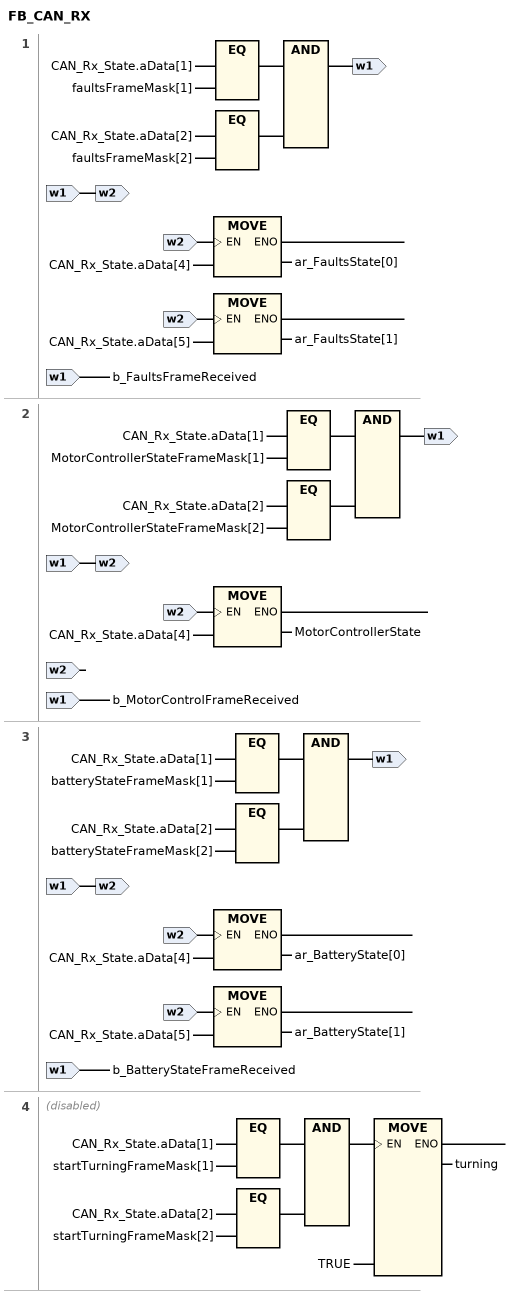
// NETWORK 1
_w1 := CAN_Rx_State.aData[1] = faultsFrameMask[1] AND CAN_Rx_State.aData[2] = faultsFrameMask[2];
_rt1(CLK := _w1);
IF _rt1.Q THEN ar_FaultsState[0] := CAN_Rx_State.aData[4]; END_IF
_rt2(CLK := _w1);
IF _rt2.Q THEN ar_FaultsState[1] := CAN_Rx_State.aData[5]; END_IF
b_FaultsFrameReceived := _w1;

// NETWORK 2
_w2 := CAN_Rx_State.aData[1] = MotorControllerStateFrameMask[1] AND CAN_Rx_State.aData[2] = MotorControllerStateFrameMask[2];
_rt3(CLK := _w2);
IF _rt3.Q THEN MotorControllerState := CAN_Rx_State.aData[4]; END_IF
b_MotorControlFrameReceived := _w2;

// NETWORK 3
_w3 := CAN_Rx_State.aData[1] = batteryStateFrameMask[1] AND CAN_Rx_State.aData[2] = batteryStateFrameMask[2];
_rt4(CLK := _w3);
IF _rt4.Q THEN ar_BatteryState[0] := CAN_Rx_State.aData[4]; END_IF
_rt5(CLK := _w3);
IF _rt5.Q THEN ar_BatteryState[1] := CAN_Rx_State.aData[5]; END_IF
b_BatteryStateFrameReceived := _w3;

// NETWORK 4 (disabled)
// _rt6(CLK := CAN_Rx_State.aData[1] = startTurningFrameMask[1] AND CAN_Rx_State.aData[2] = startTurningFrameMask[2]);
// IF _rt6.Q THEN turning := TRUE; END_IF

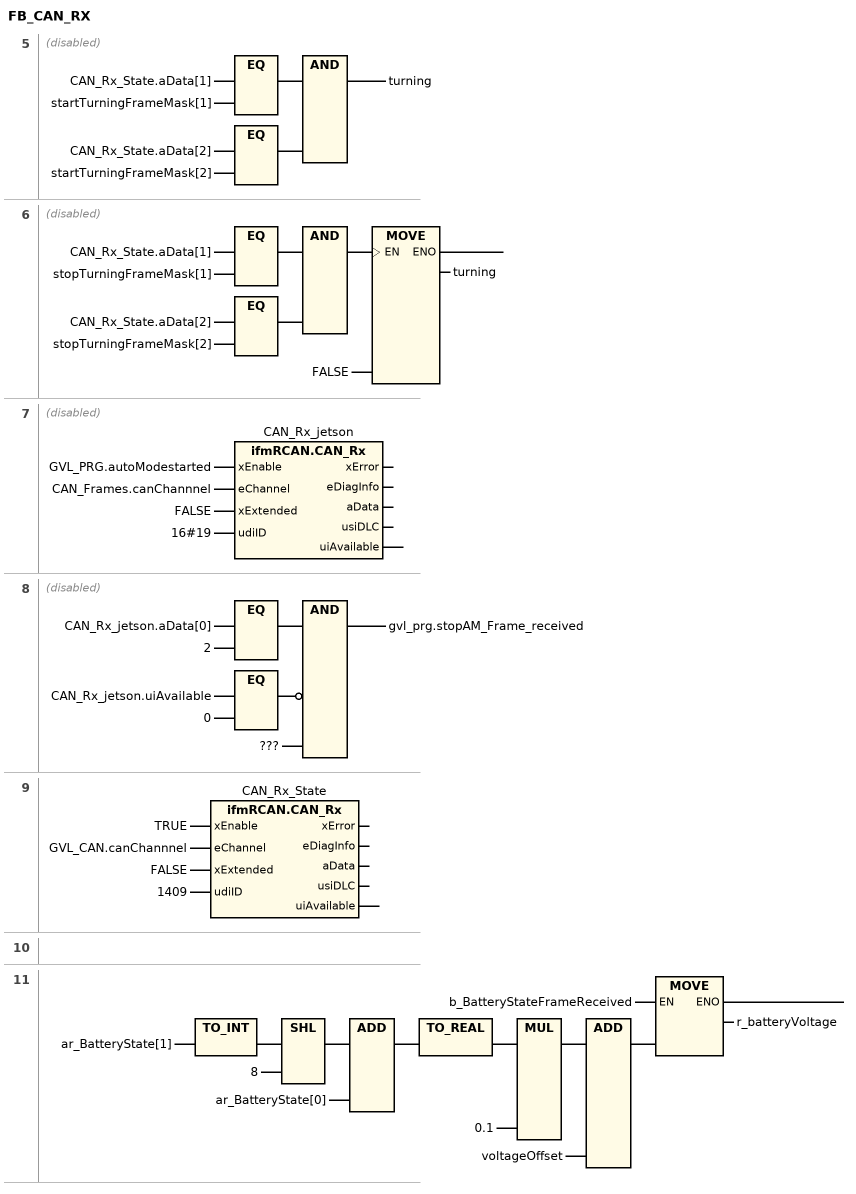
// NETWORK 5 (disabled)
// turning := CAN_Rx_State.aData[1] = startTurningFrameMask[1] AND CAN_Rx_State.aData[2] = startTurningFrameMask[2];

// NETWORK 6 (disabled)
// _rt7(CLK := CAN_Rx_State.aData[1] = stopTurningFrameMask[1] AND CAN_Rx_State.aData[2] = stopTurningFrameMask[2]);
// IF _rt7.Q THEN turning := FALSE; END_IF

// NETWORK 7 (disabled)
// CAN_Rx_jetson(
//     xEnable := GVL_PRG.autoModestarted,
//     eChannel := CAN_Frames.canChannnel,
//     xExtended := FALSE,
//     udiID := 16#19); // ifmRCAN.CAN_Rx

// NETWORK 8 (disabled)
// gvl_prg.stopAM_Frame_received := CAN_Rx_jetson.aData[0] = 2 AND NOT (CAN_Rx_jetson.uiAvailable = 0) AND ???;

// NETWORK 9
CAN_Rx_State(xEnable := TRUE, eChannel := GVL_CAN.canChannnel, xExtended := FALSE, udiID := 1409); // ifmRCAN.CAN_Rx

// NETWORK 10

// NETWORK 11
IF b_BatteryStateFrameReceived THEN
    r_batteryVoltage := TO_REAL(SHL(TO_INT(ar_BatteryState[1]), 8) + ar_BatteryState[0]) * 0.1 + voltageOffset;
END_IF

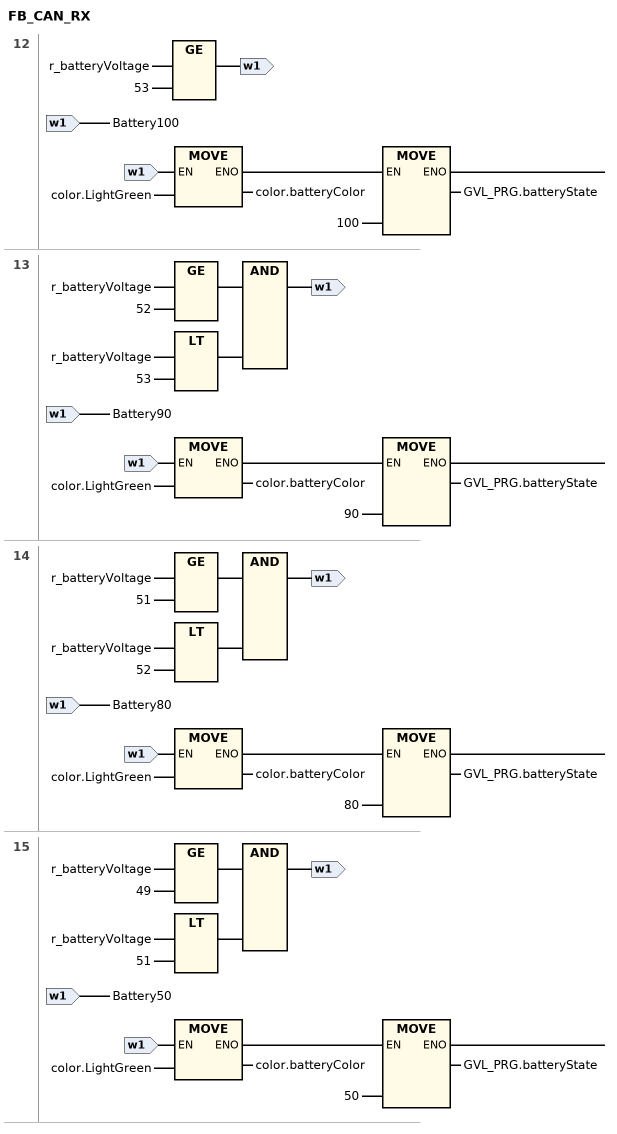
// NETWORK 12
_w4 := r_batteryVoltage >= 53;
Battery100 := _w4;
IF _w4 THEN color.batteryColor := color.LightGreen; END_IF
IF _w4 THEN GVL_PRG.batteryState := 100; END_IF

// NETWORK 13
_w5 := r_batteryVoltage >= 52 AND r_batteryVoltage < 53;
Battery90 := _w5;
IF _w5 THEN color.batteryColor := color.LightGreen; END_IF
IF _w5 THEN GVL_PRG.batteryState := 90; END_IF

// NETWORK 14
_w6 := r_batteryVoltage >= 51 AND r_batteryVoltage < 52;
Battery80 := _w6;
IF _w6 THEN color.batteryColor := color.LightGreen; END_IF
IF _w6 THEN GVL_PRG.batteryState := 80; END_IF

// NETWORK 15
_w7 := r_batteryVoltage >= 49 AND r_batteryVoltage < 51;
Battery50 := _w7;
IF _w7 THEN color.batteryColor := color.LightGreen; END_IF
IF _w7 THEN GVL_PRG.batteryState := 50; END_IF

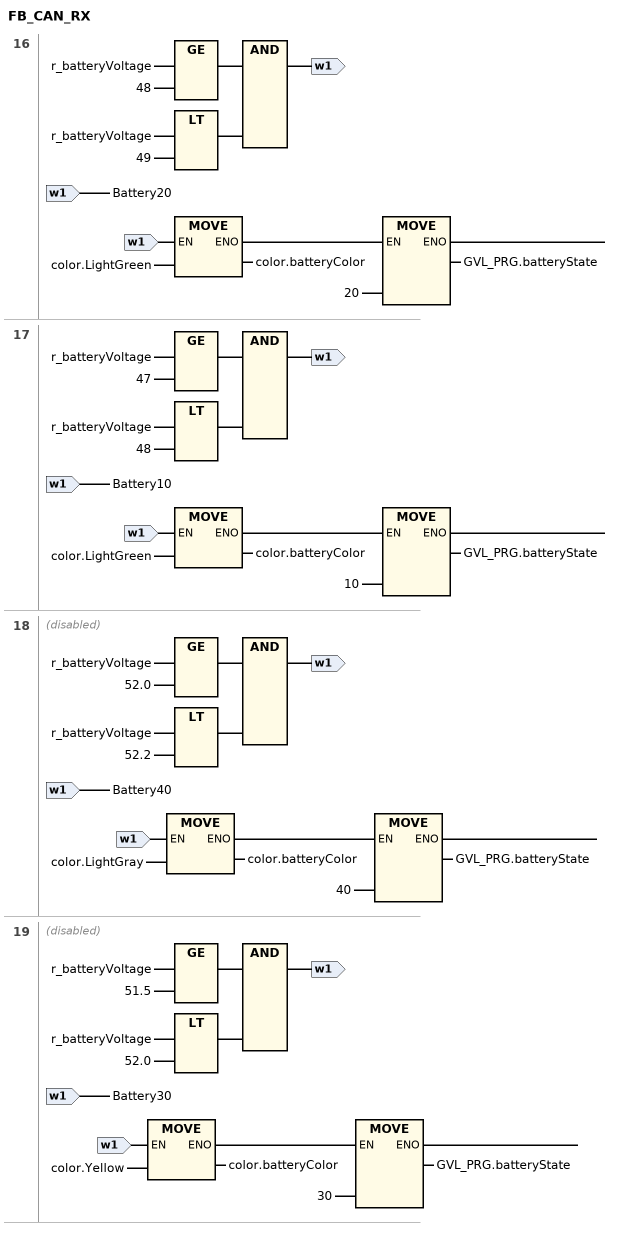
// NETWORK 16
_w8 := r_batteryVoltage >= 48 AND r_batteryVoltage < 49;
Battery20 := _w8;
IF _w8 THEN color.batteryColor := color.LightGreen; END_IF
IF _w8 THEN GVL_PRG.batteryState := 20; END_IF

// NETWORK 17
_w9 := r_batteryVoltage >= 47 AND r_batteryVoltage < 48;
Battery10 := _w9;
IF _w9 THEN color.batteryColor := color.LightGreen; END_IF
IF _w9 THEN GVL_PRG.batteryState := 10; END_IF

// NETWORK 18 (disabled)
// _w10 := r_batteryVoltage >= 52.0 AND r_batteryVoltage < 52.2;
// Battery40 := _w10;
// IF _w10 THEN color.batteryColor := color.LightGray; END_IF
// IF _w10 THEN GVL_PRG.batteryState := 40; END_IF

// NETWORK 19 (disabled)
// _w11 := r_batteryVoltage >= 51.5 AND r_batteryVoltage < 52.0;
// Battery30 := _w11;
// IF _w11 THEN color.batteryColor := color.Yellow; END_IF
// IF _w11 THEN GVL_PRG.batteryState := 30; END_IF

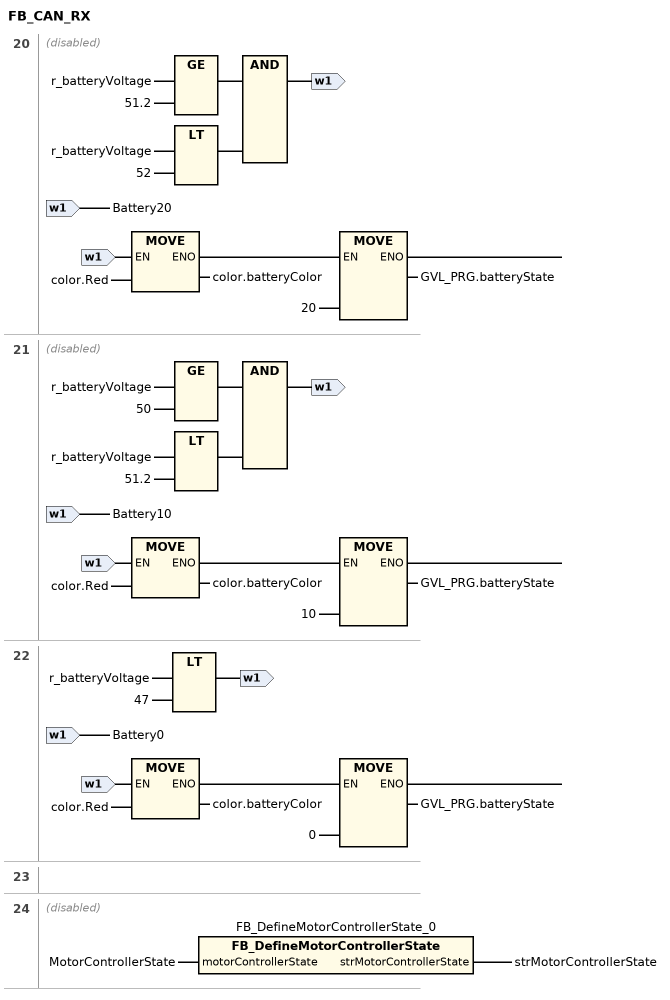
// NETWORK 20 (disabled)
// _w12 := r_batteryVoltage >= 51.2 AND r_batteryVoltage < 52;
// Battery20 := _w12;
// IF _w12 THEN color.batteryColor := color.Red; END_IF
// IF _w12 THEN GVL_PRG.batteryState := 20; END_IF

// NETWORK 21 (disabled)
// _w13 := r_batteryVoltage >= 50 AND r_batteryVoltage < 51.2;
// Battery10 := _w13;
// IF _w13 THEN color.batteryColor := color.Red; END_IF
// IF _w13 THEN GVL_PRG.batteryState := 10; END_IF

// NETWORK 22
_w14 := r_batteryVoltage < 47;
Battery0 := _w14;
IF _w14 THEN color.batteryColor := color.Red; END_IF
IF _w14 THEN GVL_PRG.batteryState := 0; END_IF

// NETWORK 23

// NETWORK 24 (disabled)
// FB_DefineMotorControllerState_0(motorControllerState := MotorControllerState); // FB_DefineMotorControllerState
// strMotorControllerState := FB_DefineMotorControllerState_0.strMotorControllerState;

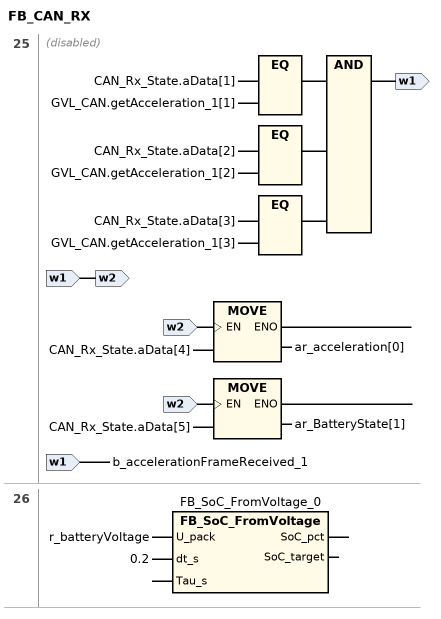
// NETWORK 25 (disabled)
// _w15 := CAN_Rx_State.aData[1] = GVL_CAN.getAcceleration_1[1] AND CAN_Rx_State.aData[2] = GVL_CAN.getAcceleration_1[2] AND CAN_Rx_State.aData[3] = GVL_CAN.getAcceleration_1[3];
// _rt8(CLK := _w15);
// IF _rt8.Q THEN ar_acceleration[0] := CAN_Rx_State.aData[4]; END_IF
// _rt9(CLK := _w15);
// IF _rt9.Q THEN ar_BatteryState[1] := CAN_Rx_State.aData[5]; END_IF
// b_accelerationFrameReceived_1 := _w15;

// NETWORK 26
FB_SoC_FromVoltage_0(U_pack := r_batteryVoltage, dt_s := 0.2); // FB_SoC_FromVoltage

END_FUNCTION_BLOCK

// Device/Application/FBs/FB_DefineMotorControllerState
FUNCTION_BLOCK FB_DefineMotorControllerState
VAR_INPUT
	motorControllerState: BYTE;
END_VAR
VAR_OUTPUT
	strMotorControllerState: STRING(100);
END_VAR
VAR
	FB_ByteToBoolArray_MotorControl: FB_ByteToBoolArray;
END_VAR

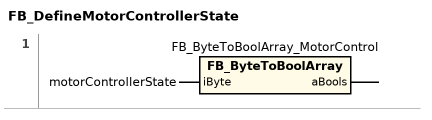
// NETWORK 1
FB_ByteToBoolArray_MotorControl(iByte := motorControllerState); // FB_ByteToBoolArray

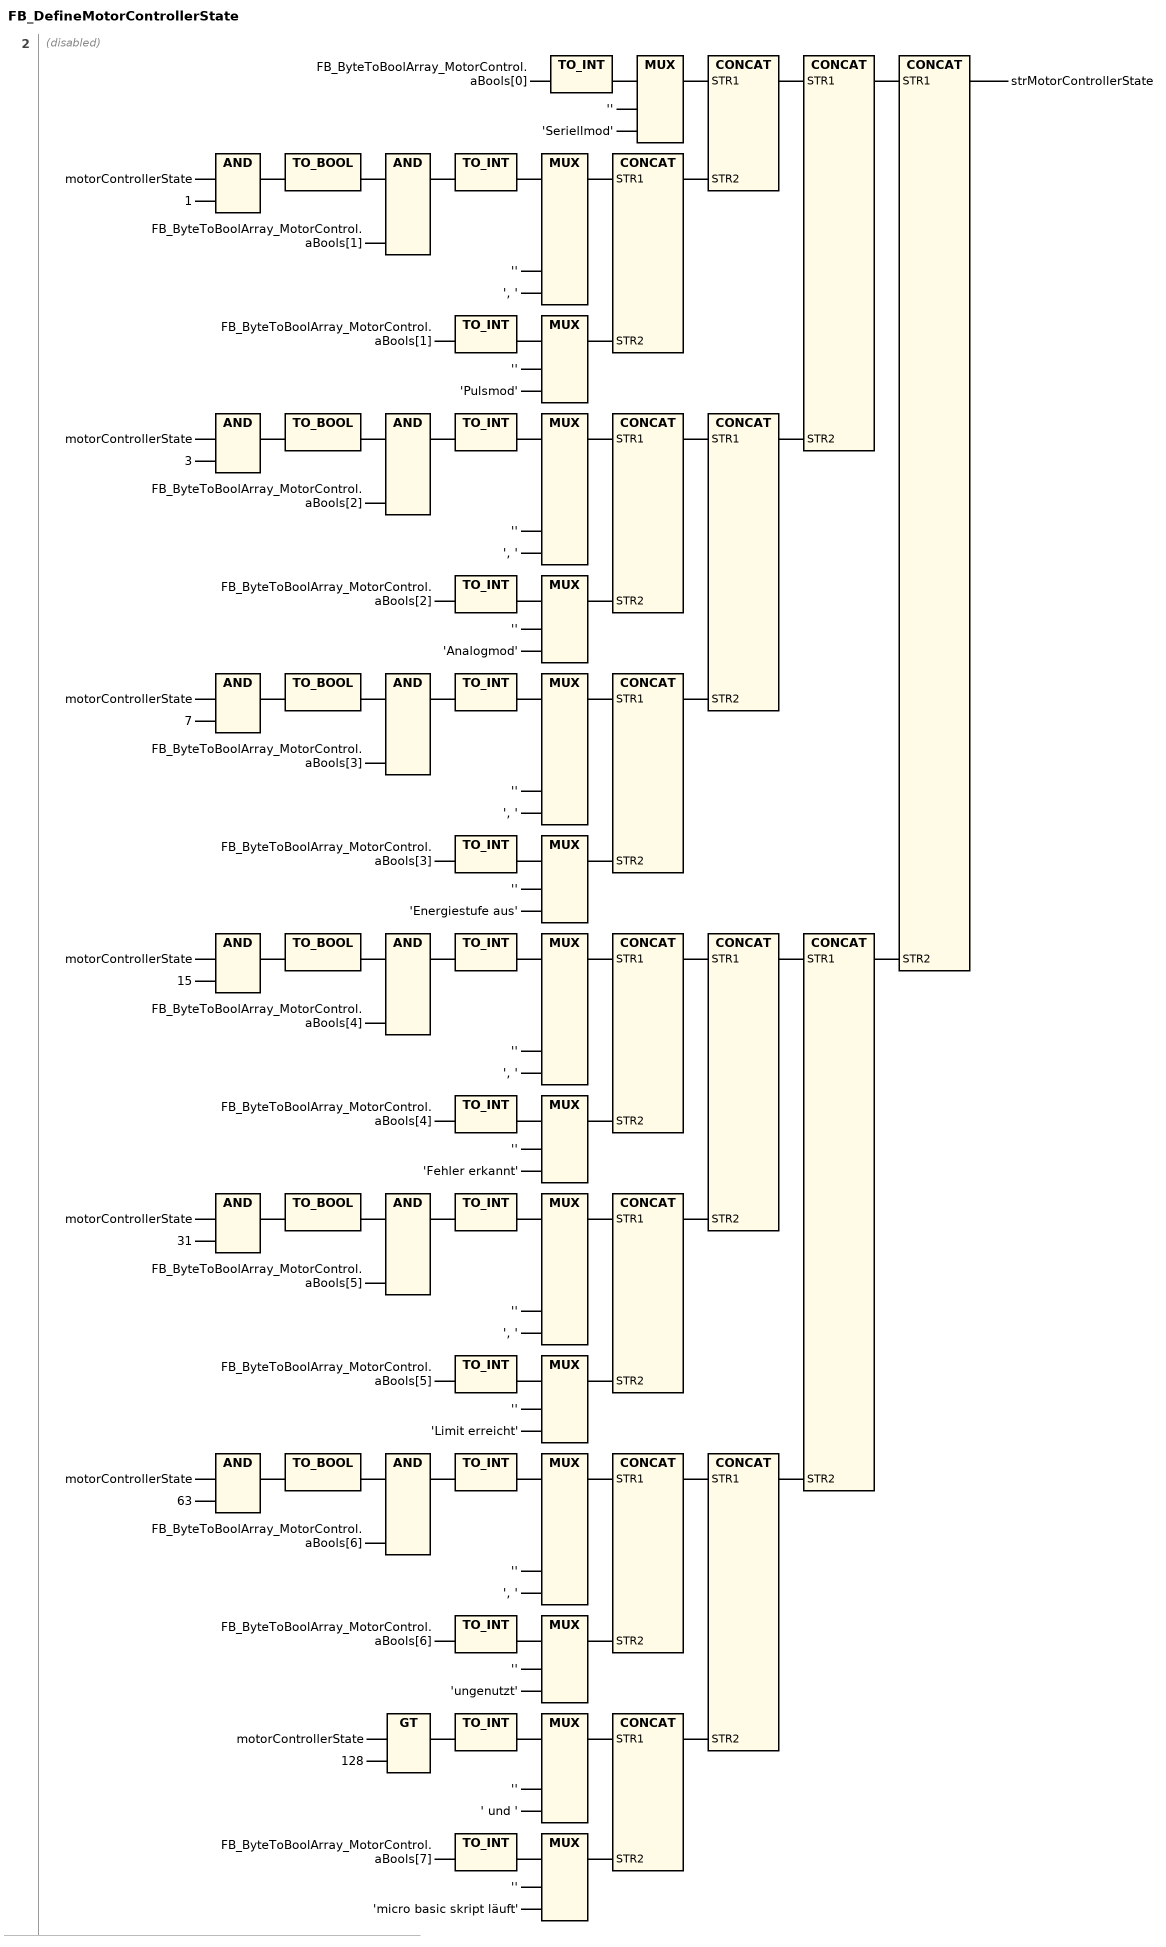
// NETWORK 2 (disabled)
// strMotorControllerState := CONCAT(STR1 := CONCAT(STR1 := CONCAT(STR1 := MUX(TO_INT(FB_ByteToBoolArray_MotorControl.aBools[0]), '', 'Seriellmod'), STR2 := CONCAT(STR1 := MUX(TO_INT(TO_BOOL(motorControllerState AND 1) AND FB_ByteToBoolArray_MotorControl.aBools[1]), '', ', '), STR2 := MUX(TO_INT(FB_ByteToBoolArray_MotorControl.aBools[1]), '', 'Pulsmod'))), STR2 := CONCAT(STR1 := CONCAT(STR1 := MUX(TO_INT(TO_BOOL(motorControllerState AND 3) AND FB_ByteToBoolArray_MotorControl.aBools[2]), '', ', '), STR2 := MUX(TO_INT(FB_ByteToBoolArray_MotorControl.aBools[2]), '', 'Analogmod')), STR2 := CONCAT(STR1 := MUX(TO_INT(TO_BOOL(motorControllerState AND 7) AND FB_ByteToBoolArray_MotorControl.aBools[3]), '', ', '), STR2 := MUX(TO_INT(FB_ByteToBoolArray_MotorControl.aBools[3]), '', 'Energiestufe aus')))), STR2 := CONCAT(STR1 := CONCAT(STR1 := CONCAT(STR1 := MUX(TO_INT(TO_BOOL(motorControllerState AND 15) AND FB_ByteToBoolArray_MotorControl.aBools[4]), '', ', '), STR2 := MUX(TO_INT(FB_ByteToBoolArray_MotorControl.aBools[4]), '', 'Fehler erkannt')), STR2 := CONCAT(STR1 := MUX(TO_INT(TO_BOOL(motorControllerState AND 31) AND FB_ByteToBoolArray_MotorControl.aBools[5]), '', ', '), STR2 := MUX(TO_INT(FB_ByteToBoolArray_MotorControl.aBools[5]), '', 'Limit erreicht'))), STR2 := CONCAT(STR1 := CONCAT(STR1 := MUX(TO_INT(TO_BOOL(motorControllerState AND 63) AND FB_ByteToBoolArray_MotorControl.aBools[6]), '', ', '), STR2 := MUX(TO_INT(FB_ByteToBoolArray_MotorControl.aBools[6]), '', 'ungenutzt')), STR2 := CONCAT(STR1 := MUX(TO_INT(motorControllerState > 128), '', ' und '), STR2 := MUX(TO_INT(FB_ByteToBoolArray_MotorControl.aBools[7]), '', 'micro basic skript läuft')))));

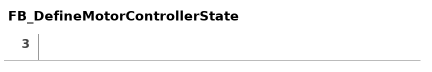
// NETWORK 3

END_FUNCTION_BLOCK

// Device/Application/FBs/Paramater/FB_ByteToBoolArray
// Der Code, um das BYTE in ein BOOL-ARRAY zu zerlegen
FUNCTION_BLOCK FB_ByteToBoolArray
VAR_INPUT
    iByte : BYTE;  // Eingangs-Byte
END_VAR

VAR_OUTPUT
    aBools : ARRAY[0..7] OF BOOL;  // Ausgangs-Array von BOOLs
	
END_VAR

VAR
    i : INT;
	byteArrayForMasking: ARRAY[0..7] OF BYTE :=[1,2,4,8,16,32,64,128];
END_VAR

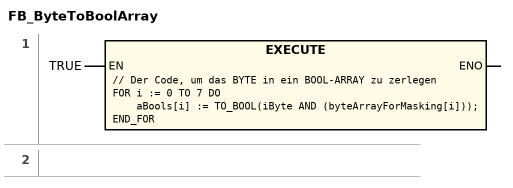
// NETWORK 1
// Der Code, um das BYTE in ein BOOL-ARRAY zu zerlegen
FOR i := 0 TO 7 DO
    aBools[i] := TO_BOOL(iByte AND (byteArrayForMasking[i]));
END_FOR

// NETWORK 2

END_FUNCTION_BLOCK

// Device/Application/FBs/Roboter_States/FB_SoC_FromVoltage
(*
    FB_SoC_FromVoltage
    - Converts LiFePO4 battery pack voltage into a % SoC value.
    - Uses a piecewise mapping with a flat plateau (49–51 V = 50 %).
    - Applies exponential smoothing (EWMA) to avoid jumps from load changes.
*)

FUNCTION_BLOCK FB_SoC_FromVoltage
VAR_INPUT
    U_pack     : REAL;    // Battery pack voltage in Volts
    dt_s       : REAL;    // Cycle time in seconds (e.g. 0.02 for 20 ms task)
    Tau_s      : REAL := 5.0; // Smoothing time constant in seconds
END_VAR
VAR_OUTPUT
    SoC_pct    : REAL;    // Smoothed State of Charge in %
    SoC_target : LREAL;    // Raw target SoC (before smoothing) in %
END_VAR
VAR
    alpha      : REAL;    // Smoothing coefficient
END_VAR

// Single-line smooth SoC from voltage (LiFePO4), scaled 0..100 %
// Smooth SoC 0..100% from voltage, no IF; anchors: 48V=10%, 50.5V=50%, 53V=90%, 54.7V=100%
SoC_target := MAX(0.0, MIN(100.0,
    10.0 + 90.0 * (
        (1.0/(1.0 + EXP(-0.75058543 * (U_pack - 50.5)))   // L(U)
        - 1.0/(1.0 + EXP(-0.75058543 * (48.0   - 50.5))))  // L(48)
        /
        (1.0/(1.0 + EXP(-0.75058543 * (54.7   - 50.5)))    // L(54.7)
        - 1.0/(1.0 + EXP(-0.75058543 * (48.0   - 50.5))))  // L(48)
    )
));

END_FUNCTION_BLOCK

// Project Information/GetCompany
// This function has been automatically generated from the project information.
{attribute 'signature_flag' := '1073741824'}
{attribute 'register_in_runtime'}
FUNCTION GetCompany : WSTRING
VAR_INPUT
	
END_VAR

GetCompany := "ifm electronic";

END_FUNCTION

// Project Information/GetTitle
// This function has been automatically generated from the project information.
{attribute 'signature_flag' := '1073741824'}
{attribute 'register_in_runtime'}
FUNCTION GetTitle : WSTRING
VAR_INPUT
	
END_VAR

GetTitle := "ifm ecomatDisplay 4.3$" 64bit with Keypad";

END_FUNCTION

// Project Information/GetVersion
// This function has been automatically generated from the project information.
{attribute 'signature_flag' := '1073741824'}
{attribute 'register_in_runtime'}
FUNCTION GetVersion : VERSION
VAR_INPUT
	
END_VAR

GetVersion.uiMajor := 4;
GetVersion.uiMinor := 0;
GetVersion.uiServicePack := 0;
GetVersion.uiPatch := 0;

END_FUNCTION

// Project Information/GetTextProperty
// This function has been automatically generated from the project information.
{attribute 'signature_flag' := '1073741824'}
{attribute 'register_in_runtime'}
FUNCTION GetTextProperty : WSTRING
VAR_INPUT
	stKey: WSTRING;
END_VAR

IF stKey = "Author" THEN
	GetTextProperty := "ifm electronic";
ELSIF stKey = "Company" THEN
	GetTextProperty := "ifm electronic";
ELSIF stKey = "CompiledLibraryCompatibilityVersion" THEN
	GetTextProperty := "CODESYS V3.5 SP16 Patch 5";
ELSIF stKey = "Description" THEN
	GetTextProperty := "Project template for 4.3$" ifm ecomat display  device with keypad.";
ELSIF stKey = "Project" THEN
	GetTextProperty := "ecomatDisplaytestIn2001";
ELSIF stKey = "Title" THEN
	GetTextProperty := "ifm ecomatDisplay 4.3$" 64bit with Keypad";
ELSE
	GetTextProperty := "";
END_IF

END_FUNCTION

// Project Information/GetTextProperty2
// This function has been automatically generated from the project information.
{attribute 'signature_flag' := '1073741824'}
{attribute 'register_in_runtime'}
FUNCTION GetTextProperty2 : POINTER TO WSTRING
VAR_INPUT
	stKey: WSTRING;
END_VAR

IF stKey = "Author" THEN
	GetTextProperty2 := ADR("ifm electronic");
ELSIF stKey = "Company" THEN
	GetTextProperty2 := ADR("ifm electronic");
ELSIF stKey = "CompiledLibraryCompatibilityVersion" THEN
	GetTextProperty2 := ADR("CODESYS V3.5 SP16 Patch 5");
ELSIF stKey = "Description" THEN
	GetTextProperty2 := ADR("Project template for 4.3$" ifm ecomat display  device with keypad.");
ELSIF stKey = "Project" THEN
	GetTextProperty2 := ADR("ecomatDisplaytestIn2001");
ELSIF stKey = "Title" THEN
	GetTextProperty2 := ADR("ifm ecomatDisplay 4.3$" 64bit with Keypad");
ELSE
	GetTextProperty2 := ADR("");
END_IF

END_FUNCTION

// Project Information/GetNumberProperty
// This function has been automatically generated from the project information.
{attribute 'signature_flag' := '1073741824'}
{attribute 'register_in_runtime'}
FUNCTION GetNumberProperty : DINT
VAR_INPUT
	stKey: WSTRING;
END_VAR

GetNumberProperty := 0;

END_FUNCTION

// Project Information/GetBooleanProperty
// This function has been automatically generated from the project information.
{attribute 'signature_flag' := '1073741824'}
{attribute 'register_in_runtime'}
FUNCTION GetBooleanProperty : BOOL
VAR_INPUT
	stKey: WSTRING;
END_VAR

IF stKey = "Released" THEN
	GetBooleanProperty := FALSE;
ELSE
	GetBooleanProperty := FALSE;
END_IF

END_FUNCTION

// Project Information/GetVersionProperty
// This function has been automatically generated from the project information.
{attribute 'signature_flag' := '1073741824'}
{attribute 'register_in_runtime'}
FUNCTION GetVersionProperty : VERSION
VAR_INPUT
	stKey: WSTRING;
END_VAR

IF stKey = "Version" THEN
	GetVersionProperty.uiMajor := 4;
	GetVersionProperty.uiMinor := 0;
	GetVersionProperty.uiServicePack := 0;
	GetVersionProperty.uiPatch := 0;
ELSE
	GetVersionProperty.uiMajor := 0;
	GetVersionProperty.uiMinor := 0;
	GetVersionProperty.uiServicePack := 0;
	GetVersionProperty.uiPatch := 0;
END_IF

END_FUNCTION

// Device/Application/functions/intToSelectOnBool
FUNCTION intToSelectOnBool
VAR_INPUT
END_VAR
VAR
END_VAR
VAR_OUTPUT
	Q0 : BOOL;
	Q1 : BOOL;
	Q2 : BOOL;
	Q3 : BOOL;
	Q4 : BOOL;
	Q5 : BOOL;
	Q6 : BOOL;
	Q7 : BOOL;
END_VAR

// NETWORK 1

END_FUNCTION

// Device/Application/functions/Stuffing_To_ArrayOfUsint
FUNCTION Stuffing_To_ArrayOfUsint : ByteArray_t
VAR_INPUT
	iData1 : USINT ;
	iData2 : USINT ;
	iData3 : USINT ;
	iData4 : USINT ;
	iData5 : USINT ;
	iData6 : USINT ;
	iData7 : USINT ;
	iData8 : USINT ;
END_VAR
VAR
	
END_VAR

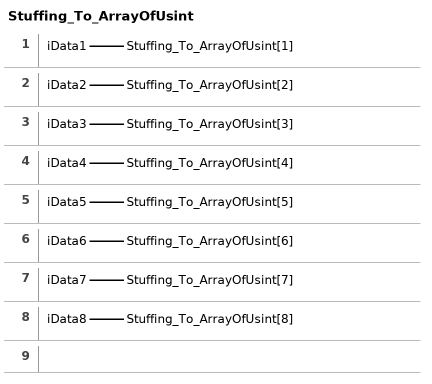
// NETWORK 1
Stuffing_To_ArrayOfUsint[1] := iData1;

// NETWORK 2
Stuffing_To_ArrayOfUsint[2] := iData2;

// NETWORK 3
Stuffing_To_ArrayOfUsint[3] := iData3;

// NETWORK 4
Stuffing_To_ArrayOfUsint[4] := iData4;

// NETWORK 5
Stuffing_To_ArrayOfUsint[5] := iData5;

// NETWORK 6
Stuffing_To_ArrayOfUsint[6] := iData6;

// NETWORK 7
Stuffing_To_ArrayOfUsint[7] := iData7;

// NETWORK 8
Stuffing_To_ArrayOfUsint[8] := iData8;

// NETWORK 9

END_FUNCTION

// Device/Application/functions/F_AnyToByte
FUNCTION F_AnyToByte : ByteArray_t
VAR_INPUT
    in_Any : ANY;                           // Eingangsvariable vom Typ ANY
END_VAR
VAR
    tempArray : ByteArray_t;                // Temporäres Array für die Rückgabe
    pSource : POINTER TO BYTE;              // Quellzeiger
    i : DINT;                               // Schleifenzähler
END_VAR

// Array initialisieren
FOR i := 0 TO 7 DO
    tempArray[i] := 0;
END_FOR

// Prüfen ob ANY-Pointer gültig ist
IF in_Any.pValue = 0 THEN
    RETURN;
END_IF

// Prüfen ob Größe im zulässigen Bereich
IF in_Any.diSize > SIZEOF(tempArray) THEN
    RETURN;
END_IF

// Zeiger auf Quelldaten setzen
pSource := in_Any.pValue;

// Bytes kopieren
FOR i := 0 TO in_Any.diSize - 1 DO
    tempArray[i] := pSource^;
    pSource := pSource + 1;
END_FOR

// Array zurückgeben
F_AnyToByte := tempArray;

END_FUNCTION

// Device/Application/Visu/Main_Site
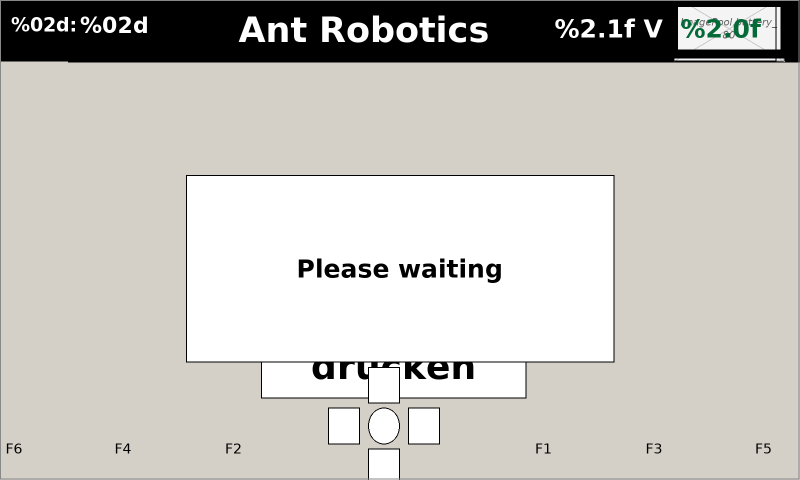
VISUALIZATION Main_Site  // 800x480
    Frame (1,62 169x230), frame switch variable: Main_FRAME_CONTROL.mainFrameId
        shows Srart_Site()
        shows Roboter_Parameter()
        shows Auto_Mode_Site()
        shows empty()
        shows NewSiteFrame()
        shows empty()
    Frame (0,-2 292x70)
        shows NewSiteFrame()
END_VISUALIZATION

// Device/Application/Visu/NewSiteFrame
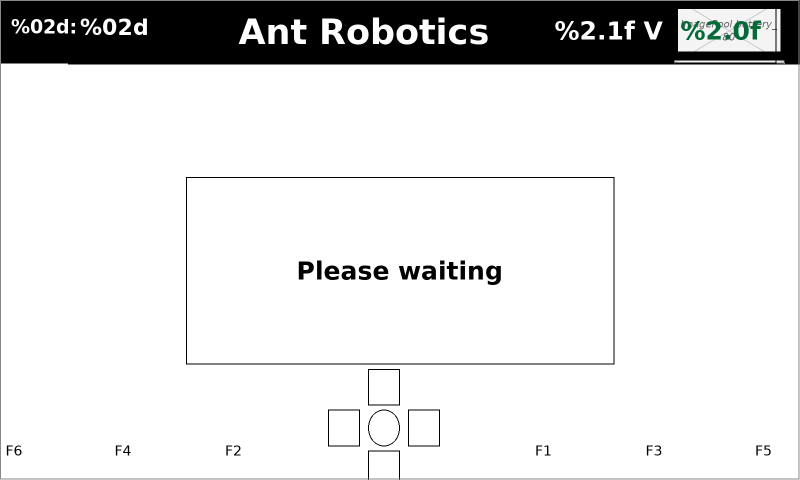
VISUALIZATION NewSiteFrame  // 800x480
    Rectangle (68,-1 592x65), "Ant Robotics"
    Rectangle (574,-2 256x66), text variable: PLC_PRG.FB_CAN_RX_0.FB_SoC_FromVoltage_0.SoC_target
    Rectangle (77,-8 70x71), "%02d", text variable: PLC_PRG.FB_HMIControl_0.stTime.uiMinute
    Rectangle (-1,-9 81x72), "%02d:", text variable: PLC_PRG.FB_HMIControl_0.stTime.uiHour
    Image (674,-2 110x65), colour toggle: TRUE, invisible if: NOT(PLC_PRG.FB_CAN_RX_0.battery90), image: ImagePool.battery_90
    Image (674,-2 110x65), colour toggle: TRUE, invisible if: NOT(PLC_PRG.FB_CAN_RX_0.battery100), image: ImagePool.battery_voll
    Image (674,-2 110x65), colour toggle: TRUE, invisible if: NOT(PLC_PRG.FB_CAN_RX_0.battery50 ), image: ImagePool.battery_50
    Image (674,-2 110x65), colour toggle: TRUE, invisible if: NOT(PLC_PRG.FB_CAN_RX_0.battery10), image: ImagePool.battery_10
    Image (674,-2 110x65), colour toggle: TRUE, invisible if: NOT(PLC_PRG.FB_CAN_RX_0.battery0), image: ImagePool.battery_0
    Image (674,-2 110x65), colour toggle: TRUE, invisible if: NOT(PLC_PRG.FB_CAN_RX_0.battery20), image: ImagePool.battery_20
    Image (674,-2 110x65), colour toggle: TRUE, invisible if: NOT(PLC_PRG.FB_CAN_RX_0.battery80), image: ImagePool.battery_80
    Rectangle (186,177 428x187), "Please waiting", invisible if: NOT(GVL_PRG.restartCan)
    Frame (-30,351 844x136), invisible if: NOT(GVL_PRG.showkeys), input disabled if: NOT(GVL_PRG.showkeys)
        shows keys_frame()
    Rectangle (666,-2 110x65), "%2.0f", text variable: PLC_PRG.FB_CAN_RX_0.FB_SoC_FromVoltage_0.SoC_target, colour toggle: PLC_PRG.FB_CAN_RX_0.FB_SoC_FromVoltage_0.SoC_target < 20, colour variable: color.batteryColor
        p2167032090: color.Blue
    Rectangle (517,-1 62x64)
    Rectangle (669,0 120x60)
    Rectangle (554,-2 110x65), "%2.1f V", text variable: PLC_PRG.FB_CAN_RX_0.r_batteryVoltage, colour toggle: PLC_PRG.FB_CAN_RX_0.FB_SoC_FromVoltage_0.SoC_target < 20, colour variable: color.batteryColor
        p2167032090: color.Blue
END_VISUALIZATION

// Device/Application/Visu/Srart_Site
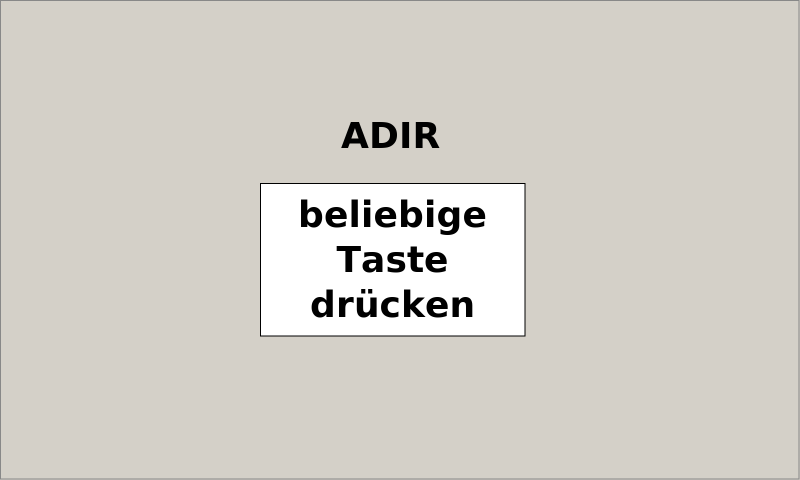
VISUALIZATION Srart_Site  // 800x480
    Rectangle (260,183 265x153), "beliebige Taste drücken"
    Rectangle (260,90 261x91), "ADIR"
    hotkey  Id=481044725760, Key=KeyName=F6, ActionToExecute=Action=ChangeLanguage=EN, VisuElemId=-1
END_VISUALIZATION

// Device/Application/Visu/Roboter_Parameter
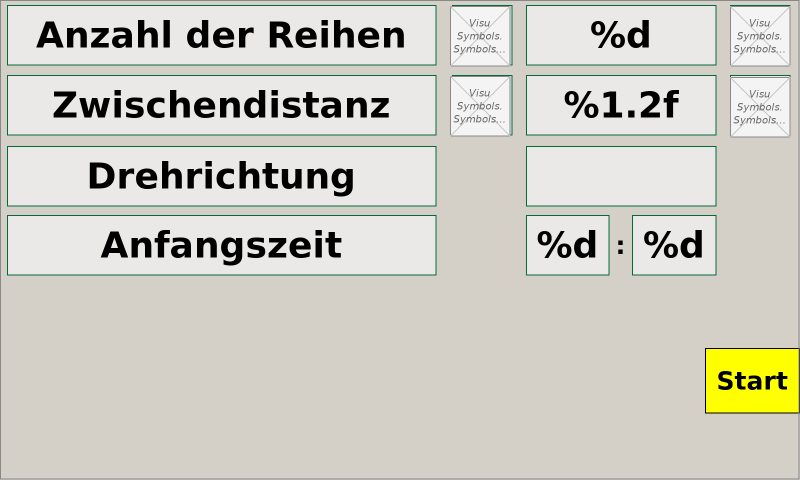
VISUALIZATION Roboter_Parameter  // 800x480
    Rectangle (705,348 95x65), "Start", colour variable: 16#FFFFFF00
        p2167032090: 16#FF00FF00
    Rectangle (452,5 60x60), colour toggle: NOT(PLC_PRG.selectedParameterIndex = 1), colour variable: 16#FF00FF00
        p2167032090: 16#FFACD5D5
    Rectangle (730,5 60x60), colour toggle: NOT(PLC_PRG.selectedParameterIndex = 1), colour variable: 16#FF00FF00
        p2167032090: 16#FFACD5D5
    Rectangle (7,5 429x60), "Anzahl der Reihen", colour toggle: NOT(PLC_PRG.selectedParameterIndex = 1), colour variable: 16#FF00FF00
        p2167032090: 16#FFACD5D5
    Rectangle (526,5 190x60), "%d", text variable: PLC_PRG.getUpdatedParameter.iCountRows, colour toggle: NOT(PLC_PRG.selectedParameterIndex = 1), colour variable: 16#FF00FF00
        p2167032090: 16#FFACD5D5
    Rectangle (7,146 429x60), "Drehrichtung", colour toggle: NOT(PLC_PRG.selectedParameterIndex = 3), colour variable: 16#FF00FF00
        p2167032090: 16#FFACD5D5
    Rectangle (526,146 190x60), text variable: PLC_PRG.getUpdatedParameter.strRowsDirection, colour toggle: NOT(PLC_PRG.selectedParameterIndex = 3), text list: 'SwitchKeys', text index: PLC_PRG.getUpdatedParameter.bRowsDirection, colour variable: 16#FF00FF00
        p2167032090: 16#FFACD5D5
    Rectangle (452,75 60x60), colour toggle: NOT(PLC_PRG.selectedParameterIndex = 2), colour variable: 16#FF00FF00
        p2167032090: 16#FFACD5D5
    Rectangle (730,75 60x60), colour toggle: NOT(PLC_PRG.selectedParameterIndex = 2), colour variable: 16#FF00FF00
        p2167032090: 16#FFACD5D5
    Rectangle (7,75 429x60), "Zwischendistanz", colour toggle: NOT(PLC_PRG.selectedParameterIndex = 2), colour variable: 16#FF00FF00
        p2167032090: 16#FFACD5D5
    Rectangle (526,75 190x60), "%1.2f", text variable: PLC_PRG.getUpdatedParameter.iDistanceBetweenRowsInMeter, colour toggle: NOT(PLC_PRG.selectedParameterIndex = 2), colour variable: 16#FF00FF00
        p2167032090: 16#FFACD5D5
    Image (450,76 60x60), colour toggle: NOT(PLC_PRG.selectedParameterIndex = 2), image: VisuSymbols.Symbols.ArrowBack
    Image (730,77 60x60), colour toggle: NOT(PLC_PRG.selectedParameterIndex = 2), image: VisuSymbols.Symbols.ArrowForward
    Image (730,6 60x60), colour toggle: NOT(PLC_PRG.selectedParameterIndex = 1), image: VisuSymbols.Symbols.ArrowForward
    Image (450,6 60x60), colour toggle: NOT(PLC_PRG.selectedParameterIndex = 1), image: VisuSymbols.Symbols.ArrowBack
    Rectangle (7,215 429x60), "Anfangszeit", colour toggle: NOT((PLC_PRG.selectedParameterIndex = 4) OR(PLC_PRG.selectedParameterIndex = 5)), colour variable: 16#FF00FF00
        p2167032090: 16#FFACD5D5
    Rectangle (526,215 83x60), "%d", text variable: gvl_prg.startHour, colour toggle: NOT(PLC_PRG.selectedParameterIndex = 4), colour variable: 16#FF00FF00
        p2167032090: 16#FFACD5D5
    Rectangle (632,215 84x60), "%d", text variable: gvl_prg.startMin, colour toggle: NOT(PLC_PRG.selectedParameterIndex = 5), colour variable: 16#FF00FF00
        p2167032090: 16#FFACD5D5
    Rectangle (608,215 25x60), ":"
END_VISUALIZATION

// Device/Application/Visu/Auto_Mode_Site
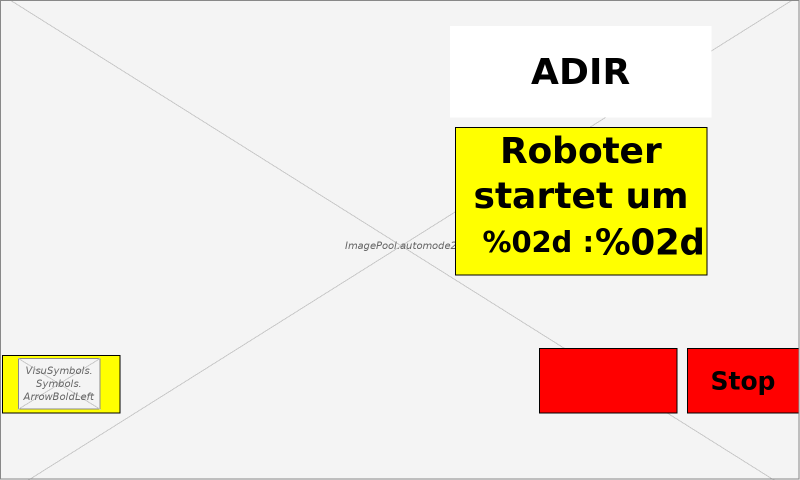
VISUALIZATION Auto_Mode_Site  // 800x480
    Image (-4,-9 810x509), image: ImagePool.automode2
    Rectangle (455,127 252x148), "Roboter ist gestartet", invisible if: NOT(GVL_PRG.autoModestarted)
    Rectangle (450,26 261x91), "ADIR"
    Rectangle (687,348 112x65), "Stop", invisible if: NOT(PLC_PRG.StopresumeButtonVisible)
    Rectangle (539,348 138x65), colour toggle: GVL_PRG.AM_Paused, invisible if: NOT(PLC_PRG.StopresumeButtonVisible), text list: 'SwitchKeys', text index: TO_INT(GVL_PRG.AM_Paused) +2, colour variable: 16#FFFF0000
        p2167032090: 16#FF00FF00
    Rectangle (455,127 252x148), "Roboter startet um", invisible if: NOT(GVL_PRG.SR_startIsKlicked.Q1)
    Rectangle (2,355 118x58)
    Image (18,358 82x51), image: VisuSymbols.Symbols.ArrowBoldLeft
    Rectangle (592,209 112x66), "%02d", text variable: gvl_prg.startMin, invisible if: NOT(GVL_PRG.SR_startIsKlicked.Q1)
    Rectangle (462,209 135x66), "%02d :", text variable: gvl_prg.startHour, invisible if: NOT(GVL_PRG.SR_startIsKlicked.Q1)
END_VISUALIZATION

// Device/Application/Visu/Visu_Default
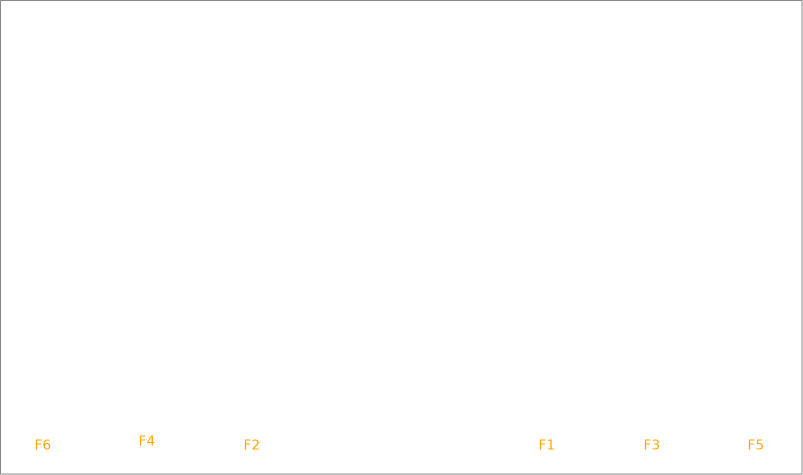
VISUALIZATION Visu_Default  // 803x475, background image ifmImagePool.DarkBg_LightKey
    Rectangle (207,415 90x60), "F2"
    Rectangle (502,415 90x60), "F1"
    Rectangle (607,415 90x60), "F3"
    Rectangle (711,415 90x60), "F5"
    Rectangle (102,411 90x60), "F4"
    Rectangle (-2,415 90x60), "F6"
END_VISUALIZATION

// Device/Application/Visu/keys_frame
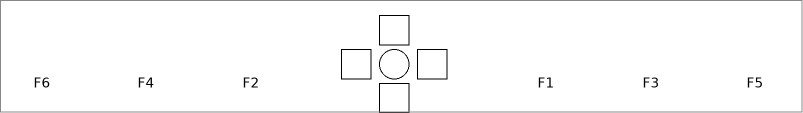
VISUALIZATION keys_frame  // 803x113
    Rectangle (206,53 90x60), "F2", invisible if: NOT(GVL_PRG.showkeys), input disabled if: NOT(GVL_PRG.showkeys)
        tap GVL_KeyList.xF2
    Rectangle (501,53 90x60), "F1", invisible if: NOT(GVL_PRG.showkeys), input disabled if: NOT(GVL_PRG.showkeys)
        tap GVL_KeyList.xF1
    Rectangle (606,53 90x60), "F3", invisible if: NOT(GVL_PRG.showkeys), input disabled if: NOT(GVL_PRG.showkeys)
        tap GVL_KeyList.xF3
    Rectangle (710,53 90x60), "F5", invisible if: NOT(GVL_PRG.showkeys), input disabled if: NOT(GVL_PRG.showkeys)
        tap GVL_KeyList.xF5
    Rectangle (101,53 90x60), "F4", invisible if: NOT(GVL_PRG.showkeys), input disabled if: NOT(GVL_PRG.showkeys)
        tap GVL_KeyList.xF4
    Rectangle (-3,53 90x60), "F6", invisible if: NOT(GVL_PRG.showkeys), input disabled if: NOT(GVL_PRG.showkeys)
        tap GVL_KeyList.xF6
    Ellipse (379,49 30x30), invisible if: NOT(GVL_PRG.showkeys), input disabled if: NOT(GVL_PRG.showkeys)
        tap GVL_KeyList.xKey_Return
    Rectangle (417,49 30x30), invisible if: NOT(GVL_PRG.showkeys), input disabled if: NOT(GVL_PRG.showkeys)
        tap GVL_KeyList.xRight
    Rectangle (379,83 30x30), invisible if: NOT(GVL_PRG.showkeys), input disabled if: NOT(GVL_PRG.showkeys)
        tap GVL_KeyList.xDown
    Rectangle (341,49 30x30), invisible if: NOT(GVL_PRG.showkeys), input disabled if: NOT(GVL_PRG.showkeys)
        tap GVL_KeyList.xLeft
    Rectangle (379,15 30x30), invisible if: NOT(GVL_PRG.showkeys), input disabled if: NOT(GVL_PRG.showkeys)
        tap GVL_KeyList.xUp
END_VISUALIZATION

// Device/Application/Visu/empty
VISUALIZATION empty  // 1024x768
END_VISUALIZATION

(* text list TL_eKeyMapCodes (id | default)
  0 | NONE
  1 | ESCAPE
  74 | MINUS
  55 | ASTERISK
  57 | SPACE
  51 | COMMA
  98 | SLASH
  78 | PLUS
  11 | KEY_0
  2 | KEY_1
  3 | KEY_2
  4 | KEY_3
  5 | KEY_4
  6 | KEY_5
  7 | KEY_6
  8 | KEY_7
  9 | KEY_8
  10 | KEY_9
  30 | KEY_A
  48 | KEY_B
  46 | KEY_C
  32 | KEY_D
  18 | KEY_E
  33 | KEY_F
  34 | KEY_G
  35 | KEY_H
  23 | KEY_I
  36 | KEY_J
  37 | KEY_K
  38 | KEY_L
  50 | KEY_M
  49 | KEY_N
  24 | KEY_O
  25 | KEY_P
  16 | KEY_Q
  19 | KEY_R
  31 | KEY_S
  20 | KEY_T
  22 | KEY_U
  47 | KEY_V
  17 | KEY_W
  45 | KEY_X
  21 | KEY_Y
  44 | KEY_Z
  28 | KEY_RETURN
  14 | BACKSPACE
  15 | TAB
  99 | PRINT
  102 | HOME
  103 | UP
  105 | LEFT
  106 | RIGHT
  107 | END
  108 | DOWN
  110 | INSERT
  111 | DELETE
  119 | PAUSE
  59 | F1
  60 | F2
  61 | F3
  62 | F4
  63 | F5
  64 | F6
  65 | F7
  66 | F8
  67 | F9
  68 | F10
  87 | F11
  88 | F12
  82 | NUM0
  79 | NUM1
  80 | NUM2
  81 | NUM3
  75 | NUM4
  76 | NUM5
  77 | NUM6
  71 | NUM7
  72 | NUM8
  73 | NUM9
   |  *)

(* text list SwitchKeys (id | default | EN | DE)
  0 | Links | Left | Links
  1 | Rechts | Right | Rechts
  2 | Pause | Pause | Pause
  3 | Weiter | Resume | Weiter
  4 | Roboter ist gestartet | Roboter started | Roboter ist gestartet
  5 | Roboter Startet um %s |  | 
   |  |  |  *)
